Fanuc KAREL source: ka00175.KL

-- PROVISIONAL review KL for V770-1; original PC SHA256 c20660dea1012b65be36862fe450bbed97289b09324212be96f735c1ef1f8e73
-- Incomplete behavior may be omitted. Consult companion uncertainty JSON. Do not deploy.
PROGRAM KA00175
%NOLOCKGROUP
BEGIN
  -- UNRESOLVED_PC offsets 5-19; opcodes 22,22,1E
  -- UNRESOLVED_PC offsets 24-28; opcodes 7F
END KA00175
